// TwinCAT 3 PLC project Untitled1
// Title: SPF_Core
// Company: Scheugenpflug
// Author: Poschmann
// ProjectVersion: 0.1.0.0
// ProgramVersion: 3.1.4023.0
// project tree:
//   FBs/ fb_Test.TcPOU
//   Version/ Global_Version.TcGVL

// ---- Version/Global_Version.TcGVL
{attribute 'TcGenerated'}
{attribute 'no-analysis'}
{attribute 'linkalways'}
// This function has been automatically generated from the project information.
VAR_GLOBAL CONSTANT
	{attribute 'const_non_replaced'}
	stLibVersion_SPF_Core : ST_LibVersion := (iMajor := 0, iMinor := 1, iBuild := 0, iRevision := 0, nFlags := 0, sVersion := '0.1.0.0');
END_VAR

// ---- FBs/fb_Test.TcPOU
FUNCTION_BLOCK fb_Test
VAR_INPUT
END_VAR
VAR_OUTPUT
	iCount : int;
END_VAR
VAR
END_VAR

iCount := iCount + 1;

END_FUNCTION_BLOCK
